TYPE ST_HTTP_Parameter :
STRUCT
	sName	: STRING;
	sValue	: STRING;
END_STRUCT
END_TYPE

(* stored: Version 1.1.0.1, ProductVersion 3.1.4020.12
   DUT ST_HTTP_Parameter: Id {4ef22fdd-9175-491e-8825-8259613d59c9} *)
